FUNCTION CompAsIReceiver : Result
VAR_INPUT
	iSource	: I_Component;
END_VAR
VAR_OUTPUT
	iDest	: I_Receiver;
END_VAR

IF iSource = 0 THEN
	CompAsIReceiver := Err.Itf0;
	RETURN;
END_IF

IF __QUERYINTERFACE(iSource, iDest) THEN
	CompAsIReceiver := Ok;
ELSE
	CompAsIReceiver := Err.NoMatch;
END_IF

END_FUNCTION

(* stored: Version 1.1.0.1
   POU CompAsIReceiver: Id {9a02776e-f8c4-45bc-8c18-325d7f2421cf}, SpecialFunc None *)
